(* IEC 61131-3 sources: programs/VI-54/VI-54_20171205/VI-54_20171205/Stations/Screen/LseClass170718/Class/AccessControlMain (part 2) *)

  if UserIsLoggedIn then
    StrActUser.GetDataAt(pData:=#tmpActUserName[0], udSize:=StrActUser.GetLength()+1, udAt:=0);
  end_if;

  tmpPos          := 0;
  pActUser        := NIL;
  tmpUserName[0]  := 0;
  tmpNewPos       := 0;

  // Benutzername angegeben
  //-----------------------------------------------------------------------------------------
  if StrEditUserName.GetLength() then

    // Benutzername und dessen Position holen
    StrEditUserName.GetDataAt(pData:=#tmpUserName[0], udSize:=StrEditUserName.GetLength()+1, udAt:=0);
    tmpNewPos := SearchUser(pBuffer := UsersBuffer, pUserName:= #tmpUserName[0], pUser:=NIL);

    // Benutzer gefunden
    //-----------------------------------------------------------------------------------------
    if (tmpNewPos >= 0) then

      // Wenn ein USB-Stick mit einem Benutzer verknüpft werden soll, muss der Benutzer manuell eingeloggt sein
      if (LoggedInWithUsb = false) & (StrEditUsbSN.GetLength() > 0) then

        //Benutzerdaten anhand der Position holen
        pActUser := getUserToEdit(udPos:=to_udint(tmpNewPos));
        tmpOwnUser := (StrCmp(p0:=#pActUser^.aUsername[0], x1:=sizeof(pActUser^.aUsername[0]), p2:=#tmpActUserName[0], x3:=sizeof(tmpActUserName[0])));
        if (pActUser <> NIL) & ((pActUser^.usUserLevel < ActLevel) | (tmpOwnUser = 0)) then

          // Wenn dieser USB-Stick schon mit einem anderen Benutzer verknüpft ist, lösche diese Verbindung
          tmpPos := SearchUserbyUsbSN(pUser:=NIL);
          if (tmpPos >= 0) then
            // Benutzerdaten anhand der Position holen
            pOldUserSN := getUserToEdit(udPos:=to_udint(tmpPos));
            if (StrCmp(p0:=#pActUser^.USBSerial[0], x1:=sizeof(pActUser^.USBSerial[0]), p2:=#pOldUserSN^.USBSerial[0], x3:=sizeof(pOldUserSN^.USBSerial[0])) <> 0) then

              if (pOldUserSN <> NIL) & ((pOldUserSN^.usUserLevel < ActLevel) | (StrCmp(p0:=#pOldUserSN^.aUsername[0], x1:=sizeof(pOldUserSN^.aUsername[0]), p2:=#tmpActUserName[0], x3:=sizeof(tmpActUserName[0])) = 0)) then
                pOldUserSN^.USBSerial[0] := 0;
              else
                MESSAGE(dMSGNumber:=ERR_AUTHORITY_EDITUSER);
                InsertCmd(x0:=CMD_NEWWINDOW, x1:=AccessControl_MessageWindowNr, x2:=0);
                return;
              end_if;

            else
              MESSAGE(dMSGNumber:=ERR_USB_SERNUM);
              InsertCmd(x0:=CMD_NEWWINDOW, x1:=AccessControl_MessageWindowNr, x2:=0);
            end_if;

          end_if;

          // Seriennummer des USB-Sticks speichern
          StrEditUsbSN.GetDataAt(pData:=#pActUser^.USBSerial[0], udSize:=StrEditUsbSN.GetLength()+1, udAt:=0);
          refreshUserFile();

        else

          MESSAGE(dMSGNumber:=ERR_AUTHORITY_EDITUSER);
          InsertCmd(x0:=CMD_NEWWINDOW, x1:=AccessControl_MessageWindowNr, x2:=0);

        end_if;
      else

        MESSAGE(dMSGNumber:=ERR_USB_SERNUM);
        InsertCmd(x0:=CMD_NEWWINDOW, x1:=AccessControl_MessageWindowNr, x2:=0);

      end_if;

    else

      MESSAGE(dMSGNumber:=ERR_USER_NOTEXIST);
      InsertCmd(x0:=CMD_NEWWINDOW, x1:=AccessControl_MessageWindowNr, x2:=0);

    end_if;

  else

    MESSAGE(dMSGNumber:=ERR_NO_NAME);
    InsertCmd(x0:=CMD_NEWWINDOW, x1:=AccessControl_MessageWindowNr, x2:=0);

  end_if;

END_FUNCTION

FUNCTION VIRTUAL GLOBAL AccessControlMain::IF_WindowEnd
	VAR_INPUT
		whoami 	: ^_WHOAMI;
		pic 	: ^void;
	END_VAR

  // Alle Server beim Schließen eines Fensters zurücksetzen
  //-----------------------------------------------------------------------------------------
  if (whoami^.ima <> IMA_TOUCHEDITOR) then

    clearServers();

  end_if;

END_FUNCTION

FUNCTION GLOBAL AccessControlMain::DelUsbSN
  VAR
    tmpPos         : DINT;
    tmpOwnUser     : UINT;
    pActUser       : ^t_s_User;
    tmpUserName    : ARRAY[0..AccessControl_MaxUsernameLength] of CHAR;
    tmpActUserName : ARRAY[0..AccessControl_MaxUsernameLength] of CHAR;
  END_VAR

  tmpPos            := 0;
  pActUser          := NIL;
  tmpUserName[0]    := 0;
  tmpActUserName[0] := 0;

  // Benutzername angegeben
  //-----------------------------------------------------------------------------------------
  if StrEditUserName.GetLength() then

    StrEditUserName.GetDataAt(pData:=#tmpUserName[0], udSize:=StrEditUserName.GetLength()+1, udAt:=0);
    StrActUser.GetDataAt(pData:=#tmpActUserName[0], udSize:=StrActUser.GetLength()+1, udAt:=0);

    // Position des Benutzers holen
    tmpPos := SearchUser(pBuffer := UsersBuffer, pUserName:=#tmpUserName[0], pUser:=NIL);
    if (tmpPos >= 0) then

      // Benutzerdaten anhand der Position holen
      pActUser := getUserToEdit(to_udint(tmpPos));
      tmpOwnUser := (StrCmp(p0:=#tmpUserName[0], x1:=sizeof(tmpUserName[0]), p2:=#tmpActUserName[0], x3:=sizeof(tmpActUserName[0])));
      if (pActUser <> NIL) & ((tmpOwnUser) | ((tmpOwnUser = 0) & (LoggedInWithUsb = 0))) &
         (StrLen(txt:=#pActUser^.USBSerial[0], size:=sizeof(pActUser^.USBSerial[0])) <> 0) then

        // Berechtigt um diesen Benutzer zu bearbeiten bzw. den eigenen Benutzer bearbeiten
        if ((pActUser^.usUserLevel < ActLevel) | (tmpOwnUser = 0)) then
          pActUser^.USBSerial[0] := 0;
          refreshUserFile();
        else
          MESSAGE(dMSGNumber:=ERR_AUTHORITY_EDITUSER);
          InsertCmd(x0:=CMD_NEWWINDOW, x1:=AccessControl_MessageWindowNr, x2:=0);
        end_if;

      else

        MESSAGE(dMSGNumber:=ERR_DEL_USB_SERNUM);
        InsertCmd(x0:=CMD_NEWWINDOW, x1:=AccessControl_MessageWindowNr, x2:=0);

      end_if;

    else

      MESSAGE(dMSGNumber:=ERR_USER_NOTEXIST);
      InsertCmd(x0:=CMD_NEWWINDOW, x1:=AccessControl_MessageWindowNr, x2:=0);

    end_if;

  else

    MESSAGE(dMSGNumber:=ERR_NO_NAME);
    InsertCmd(x0:=CMD_NEWWINDOW, x1:=AccessControl_MessageWindowNr, x2:=0);

  end_if;

END_FUNCTION

FUNCTION VIRTUAL GLOBAL AccessControlMain::CopyUserFile::Write
	VAR_INPUT
		input (EAX) 	: DINT;
	END_VAR
	VAR_OUTPUT
		result (EAX) 	: DINT;
	END_VAR
  VAR
    tmpExtDriveLetter : ARRAY[0..AccessControl_MaxUserFilePathLength] of CHAR;
    tmpFileCpy        : DINT;
  END_VAR

	CopyUserFile := input;
	result := CopyUserFile;

  // Exportieren/Importieren der Benutzerdatei auf einen USB-Speicher
  //-----------------------------------------------------------------------------------------
  if (CopyUserFile <> 0) then

    // USB-Speichermedium auch angeschlossen?
    //-----------------------------------------------------------------------------------------
    if coDriveLetter.GetLength() then

      tmpExtDriveLetter[0] := 0;
      coDriveLetter.GetDataAt(pData:=#tmpExtDriveLetter[0], udSize:=coDriveLetter.GetLength()+1, udAt:=0);
      StrNCpy(p0:=#tmpExtDriveLetter[AccessControl_DriveLetterLength],
              x1:=sizeof(tmpExtDriveLetter[0]),
              p2:=AccessControl_UserFile,
              x3:=sizeof(_ASCII),
              ml:=AccessControl_MaxUserFilePathLength);

      // Bestehende Datei der Benutzerdaten auf entsprechendes Laufwerk kopieren
      //-----------------------------------------------------------------------------------------
      if (CopyUserFile > 0) then
        // Exportieren der Benutzerdatei auf einen USB-Speicher
        tmpFileCpy := coFileSys.FileCopy(pSource:=AccessControl_InitDriveLetter, pDest:=#tmpExtDriveLetter[0], udOption:=0);
      elsif (CopyUserFile < 0) then
        // Importieren der Benutzerdatei von einem USB-Speicher
        tmpFileCpy := coFileSys.FileCopy(pSource:=#tmpExtDriveLetter[0], pDest:=AccessControl_InitDriveLetter, udOption:=0);
      end_if;

      // Kopieren der Benutzerdaten erfolgreich?
      if (tmpFileCpy <> 0) then
        MESSAGE(dMSGNumber:=ERR_COPYUSERS);
        InsertCmd(x0:=CMD_NEWWINDOW, x1:=AccessControl_MessageWindowNr, x2:=0);
        if IsCon_coSystemLogging = TRUE then
          coSystemLogging.LogEventText("AccessControlMain::CopyUserFile::Write(): Kopieren der Benutzerdaten fehlgeschlagen" );
        end_if;
      elsif (CopyUserFile > 0) & (tmpFileCpy = 0) then
        MESSAGE(dMSGNumber:=MSG_EXPORT_USERS_OK);
        InsertCmd(x0:=CMD_NEWWINDOW, x1:=AccessControl_MessageWindowNr, x2:=0);
      elsif (CopyUserFile < 0) & (tmpFileCpy = 0) then
        MESSAGE(dMSGNumber:=MSG_IMPORT_USERS_OK);
        InsertCmd(x0:=CMD_NEWWINDOW, x1:=AccessControl_MessageWindowNr, x2:=0);
      end_if;

    else

      MESSAGE(dMSGNumber:=ERR_NO_DRIVE);
      InsertCmd(x0:=CMD_NEWWINDOW, x1:=AccessControl_MessageWindowNr, x2:=0);

    end_if;

    // Server zurücksetzen
    CopyUserFile := 0;

  end_if;

END_FUNCTION

FUNCTION AccessControlMain::closeScreen

  // Benutzer befindet sich auf einem Screen, ohne korrekte Zugangsberechtigung
  if (bCloseScreen = true & (bdAccessConfig.IgnoreScreenAccess = 0)) then

    // Kehre zum Start-Bildschirm zurück
    InsertCmd(x0:=CMD_NEWPICTURE, x1:=coGlobal.GetStartPicture(), x2:=0);
    bCloseScreen := false;

  end_if;

END_FUNCTION

FUNCTION GLOBAL AccessControlMain::CreateAdmin
	VAR_INPUT
		pUsername 	: ^CHAR;
		pPassword 	: ^CHAR;
		usLevel 	: USINT;
	END_VAR
	VAR_OUTPUT
		bSuccessful 	: BOOL;
	END_VAR

  //Rückgabewert initialisieren
  bSuccessful := FALSE;

  if StandardUser = NIL then

    StandardUser$^void := coSystem.Malloc(sizeof(t_s_VKUser));
    StandardUser^.pNext := NIL;

  end_if;

  //Benutzerdaten gültig?
  if (pUsername <> NIL) & (pPassword <> NIL) & (usLevel <> NIL) then

    StrNCpy(p0 := #StandardUser^.User.aUsername[0],
            x1 := sizeof(StandardUser^.User.aUsername[0]),
            p2 := pUsername,
            x3 := sizeof(_ASCII),
            ml := AccessControl_MaxUsernameLength);
    StrNCpy(p0 := #StandardUser^.User.aUserPassword[0],
            x1 := sizeof(StandardUser^.User.aUserPassword[0]),
            p2 := pPassword,
            x3 := sizeof(_ASCII),
            ml := AccessControl_MaxPasswordLength);
    StandardUser^.User.usUserLevel   := usLevel;
    StandardUser^.User.udUserTimeout := 0;

     bSuccessful := true;
  end_if;

END_FUNCTION

FUNCTION VIRTUAL GLOBAL AccessControlMain::IF_ChkEnable
	VAR_INPUT
		key 	: DINT;
	END_VAR
	VAR_OUTPUT
		retcode 	: BOOL;
	END_VAR

  retcode := false;

  // Zugangsebenen deaktiviert (frei zugänglich)
  //-----------------------------------------------------------------------------------------
  if (Deactivate = true) then

    retcode := true;

  // Zugangscode prüfen
  //-----------------------------------------------------------------------------------------
  elsif (ActLevel >= key) then

    retcode := true;

  end_if;

END_FUNCTION

FUNCTION GLOBAL AccessControlMain::ReloadRecipe
	VAR_INPUT
		ReadValue 	: DINT;
	END_VAR
	VAR_OUTPUT
		State 	: DINT;
	END_VAR

  if ReadValue = 1 then
    Reload := 0;
  end_if;

  State := Reload;

END_FUNCTION
